RoboDK station: HAMK_solution_python_attach_mosaic_vacuum_gripper_MG400.rdk

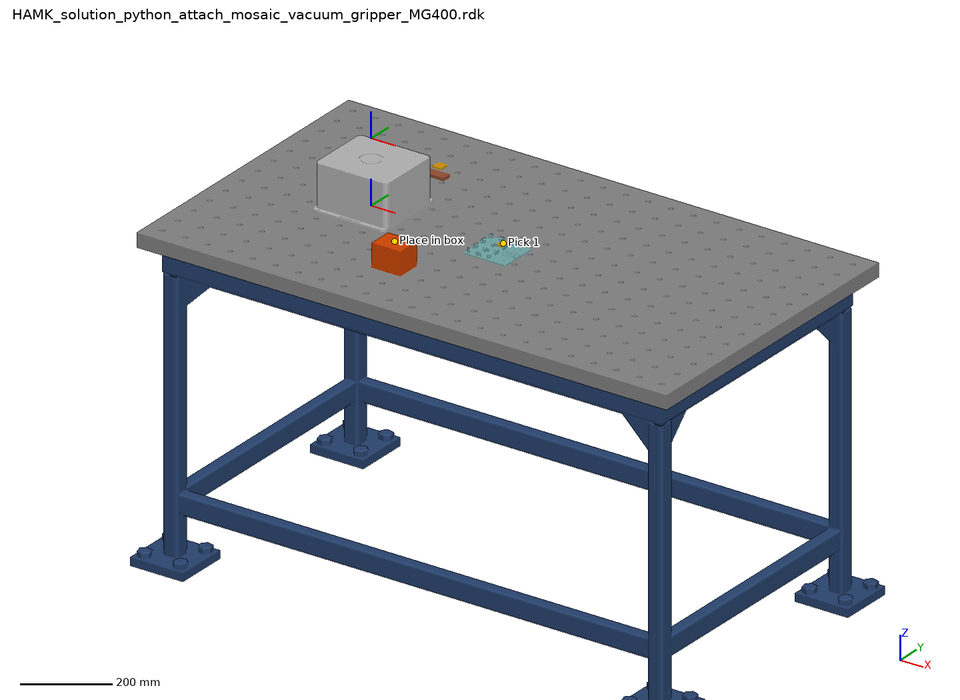
[picture v0: the station drawn from its stored meshes, robots at their saved joint values, targets as dots, program paths as lines]
Station HAMK_solution_python_attach_mosaic_vacuum_gripper_MG400 (saved by RoboDK 5.8.0). Poses are relative to the parent item; angles as X-Y-Z fixed-axis rotations.
Station parameters (name, value as stored): IO_1, 1, IO_5, 1, 1, 0, 2, 0
  - frame Dobot MG400 Base at (0, 0, 0) mm
    - robot Dobot MG400: 4 axes, payload 0.5 kg, reach 393.5 mm, repeatability 0.2 mm, weight 4 kg
        joint limits [-160, -25, -25, -360] to [160, 85, 105, 360]; home [0, 0, 0, 0]; saved at [-45.526, 49.731, 68.096, 134.474]
      - tool Suction Cup, TCP at (0, 0, -76) mm, size 42.6 x 40 x 76.8 mm
    - frame World at (0, 0, 0) mm
      - object Table 1400x800x800mm at (0, 0, 0) mm, size 1420 x 820 x 800 mm, geometry from Table-1400x800x800mm.sld
        - object HAMK logo at (360, 380, -115) mm, rotated rx 90 ry 0 rz 180 deg, size 301.4 x 100.9 x 9.4 mm, geometry from Fantastic Duup(2).stl
        - object white background at (360, 385.5, -110) mm, rotated rx 90 ry 0 rz 0 deg, size 480 x 184.8 x 2.4 mm, geometry from Fantastic Duup(3).stl
      - object Kapla wood block 0 at (0, 200, 0) mm, size 117 x 23.4 x 7.8 mm, geometry from Kapla wood block.stl
      - object Box at (176, -250, 0) mm, size 76 x 62 x 60 mm, geometry from cube.sld
      - object Mosaic tile 0 at (0, 230, 0) mm, size 24 x 24 x 4 mm, geometry from cube.sld
      - object HAMK mosaic frame at (340, -30, 0) mm, size 110 x 100 x 13 mm, geometry from pick_place_frame.stp
      - object Mosaic tile 1 at (338.5, -12, 3) mm, size 24 x 24 x 4 mm, geometry from cube.sld
  - frame RefSuctionCup at (0, 0, 161.75) mm
    - target Pick 1 (Cartesian target) at (350, 0, -154) mm; joints [0, 71.634, 64.835, 180] of Dobot MG400
    - target Place in box (Cartesian target) at (216, -220, -100) mm; joints [-45.526, 49.731, 68.096, 134.474] of Dobot MG400
  - Python program Prog0 (listed below)
  - Python program Prog1 (listed below)
  - Python program Prog3 (listed below)
  - Python program Prog4-Attach (listed below)
  - program Prog5 (1 instructions, listed below)

--- Python program Prog0 ---
# Using Python for pick and place
# Fernando Pacheco
# 2024-11
# v0: Only 2 targets, without approach. Not the right way to do

from robodk import robolink    # RoboDK API
from robodk import robomath    # Robot toolbox

# Connect to RoboDK
RDK = robolink.Robolink()

# Get the robot
# RDK.Item searches for items in the station
robot = RDK.Item('Dobot MG400', robolink.ITEM_TYPE_ROBOT)
# Get the targets
pick = RDK.Item('Pick 1')
place = RDK.Item('Place in box')

# Movements
robot.MoveJ(pick)
robot.setDO('1',1)
robot.Pause(200)
robot.MoveJ(place)
robot.setDO('1',0)

--- Python program Prog1 ---
"""
Using Python for pick and place
Fernando Pacheco
2024-11
v1: With approach positions created programmaticaly
Process:
    Locate target
    Copy it
    Paste it in the reference frame
    Change the name to approach_
    Move the target in the z-axis
"""

from robodk import robolink    # RoboDK API
from robodk import robomath    # Robot toolbox

# Connect to RoboDK
RDK = robolink.Robolink()

# Get the robot
# RDK.Item searches for items in the station
robot = RDK.Item('Dobot MG400', robolink.ITEM_TYPE_ROBOT)

# Get the reference frame
frame = RDK.Item('RefSuctionCup')

# Get the target Pick 1, copy it and create approach position
pick = RDK.Item('Pick 1')
pick.Copy() # equivalent to using CTRL+C

approach_pick = frame.Paste() # equivalent to CTRL+V
approach_pick.setName('Approach 1')
approach_pick.setPose(approach_pick.Pose()*robomath.transl(tz=80))

place = RDK.Item('Place in box')

# Movements
robot.MoveJ(approach_pick)
robot.MoveL(pick)
robot.setDO('1',1) # turn on Vacuum
robot.Pause(200)
robot.MoveL(approach_pick)
robot.MoveJ(place)
robot.setDO('1',0)
robot.setDO('2',1) # turn on Pressure
robot.Pause(200)
robot.setDO('2',0)

--- Python program Prog3 ---
"""
Using Python for pick and place
Fernando Pacheco
2024-11
v3: With more titles,
    pick and approach positions created programmaticaly
Process:
    Locate Pick 1
    Copy Pick 1
    Loop for i in range(2,num_titles+1):
        Paste Pick 1 in the reference frame
        Change the name to Pick_i
        Move Pick_i in the y-axis
    Loop for i in range(1,num_titles+1):
        Paste Pick 1 in the reference frame
        Change the name to Approach_i
        Move Approach_i in the y-axis and z-axis
"""

from robodk import robolink    # RoboDK API
from robodk import robomath    # Robot toolbox

num_titles=3 # number of mosaic titles to pick

# Connect to RoboDK
RDK = robolink.Robolink()

# Get the robot
# RDK.Item searches for items in the station
robot = RDK.Item('Dobot MG400', robolink.ITEM_TYPE_ROBOT)

# Get the reference frame
frame = RDK.Item('RefSuctionCup')

# Get the target Pick 1, copy it
pick = RDK.Item('Pick 1')
pick.Copy() # equivalent to using CTRL+C

for i in range(2, num_titles+1):
    temp = frame.Paste() # equivalent to CTRL+V
    temp.setName('Pick '+str(i))
    temp.setPose(temp.Pose()*robomath.transl(ty=-30*(i-1)))

# similar to Approach_i
for i in range(1, num_titles+1):
    temp = frame.Paste() # equivalent to CTRL+V
    temp.setName('Approach '+str(i))
    temp.setPose(temp.Pose()*robomath.transl(ty=-30*(i-1), tz=80))

place = RDK.Item('Place in box')

# Movements
for i in range(1, num_titles+1):
    approach_pick = RDK.Item('Approach '+str(i))
    pick = RDK.Item('Pick '+str(i))
    robot.MoveJ(approach_pick)
    robot.MoveL(pick)
    robot.setDO('1',1) # turn on Vacuum
    robot.Pause(200)
    robot.MoveL(approach_pick)
    robot.MoveJ(place)
    robot.setDO('1',0)
    robot.setDO('2',1) # turn on Pressure
    robot.Pause(200)
    robot.setDO('2',0)

--- Python program Prog4-Attach ---
"""
Using Python for pick and place
Fernando Pacheco
2024-12
v3: With more titles,
    pick and approach positions created programmaticaly
    include attach and detach events
Process:
    Locate Pick 1
    Copy Pick 1
    Loop for i in range(2,num_titles+1):
        Paste Pick 1 in the reference frame
        Change the name to Pick_i
        Move Pick_i in the y-axis
    Loop for i in range(1,num_titles+1):
        Paste Pick 1 in the reference frame
        Change the name to Approach_i
        Move Approach_i in the y-axis and z-axis
"""

from robodk import robolink    # RoboDK API
from robodk import robomath    # Robot toolbox

num_tiles=3 # number of mosaic titles to pick

# Connect to RoboDK
RDK = robolink.Robolink()

# Get the robot
# RDK.Item searches for items in the station
robot = RDK.Item('Dobot MG400', robolink.ITEM_TYPE_ROBOT)

# Get the reference frame
frame = RDK.Item('RefSuctionCup')

# Get the target Pick 1, copy it
pick = RDK.Item('Pick 1')
pick.Copy() # equivalent to using CTRL+C

for i in range(2, num_tiles+1):
    temp = frame.Paste() # equivalent to CTRL+V
    temp.setName('Pick '+str(i))
    temp.setPose(temp.Pose()*robomath.transl(ty=-30*(i-1)))

# similar to Approach_i
for i in range(1, num_tiles+1):
    temp = frame.Paste() # equivalent to CTRL+V
    temp.setName('Approach '+str(i))
    temp.setPose(temp.Pose()*robomath.transl(ty=-30*(i-1), tz=80))

place = RDK.Item('Place in box')

# attach and detach (only for the simulation)
tool = RDK.Item('Suction Cup')
world = RDK.Item('World')
mosaic = RDK.Item('Mosaic tile 1')
mosaic.Copy()
# then copy mosaic tiles
for i in range(2, num_tiles+1):
    temp = world.Paste() # equivalent to CTRL+V
    temp.setName('Mosaic tile '+str(i))
    temp.setPose(temp.Pose()*robomath.transl(ty=-30*(i-1)))

# Movements
for i in range(1, num_tiles+1):
    approach_pick = RDK.Item('Approach '+str(i))
    pick = RDK.Item('Pick '+str(i))
    robot.MoveJ(approach_pick)
    robot.MoveL(pick)
    tool.AttachClosest()
    robot.setDO('1',1) # turn on Vacuum
    robot.Pause(200)
    robot.MoveL(approach_pick)
    robot.MoveJ(place)
    tool.DetachAll(parent=world)
    robot.setDO('1',0)
    robot.setDO('2',1) # turn on Pressure
    robot.Pause(200)
    robot.setDO('2',0)
robot.MoveJ(approach_pick)

--- program Prog5 (robot Dobot MG400) ---
  Replace objects
